(* PLC project Unnamed, Unknown Unnamed 1 *)
(* stored: creationDateTime 2026-07-02T15:04:41, modificationDateTime 2026-07-02T15:04:41 *)

FUNCTION DIV : ANY_NUM
  VAR_INPUT
    IN1 : ANY_NUM;
    IN2 : ANY_NUM;
  END_VAR

END_FUNCTION

FUNCTION MOVE : ANY
  VAR_INPUT
    IN : ANY;
  END_VAR

END_FUNCTION

PROGRAM main
  VAR_INPUT
    S1_LiDAR_Posisi : BOOL;  (* TRUE jika LiDAR mendeteksi posisi truk sudah pas/pas di tengah. *)
    S2_LoadCell_Stable : BOOL;  (* TRUE jika pembacaan berat dari load cell sudah stabil (tidak fluktuatif). *)
    Reset_Button : BOOL;  (* Tombol untuk meriset sistem setelah truk selesai ditimbang dan keluar. *)
    LiDAR_Volume_Raw : INT;  (* Data raw volume dari LiDAR. *)
    LoadCell_Weight_Raw : INT;  (* Data raw berat dari Load Cell. *)
  END_VAR
  VAR_OUTPUT
    Sistem_Ready : BOOL;  (* Lampu indikator jembatan timbang siap menerima truk. *)
    Alarm_Posisi : BOOL;  (* Lampu/sirine jika truk berhenti di posisi yang salah. *)
    Density_Result : REAL;  (* Hasil akhir perhitungan massa jenis (p). *)
  END_VAR
  VAR
    Lock_Data : BOOL;  (* Relay internal untuk mengunci proses kalkulasi. *)
    Volume_Locked : REAL;  (* Memori untuk menyimpan data volume yang sudah dikunci. *)
    Weight_Locked : REAL;  (* Memori untuk menyimpan data berat yang sudah dikunci. *)
  END_VAR
  VAR  (* added by the conversion: wires and edge detectors of the diagram *)
    R_TRIG1 : R_TRIG;
    R_TRIG2 : R_TRIG;
  END_VAR

(* LD diagram, written out as Structured Text *)
Sistem_Ready := NOT Lock_Data;
Alarm_Posisi := NOT S1_LiDAR_Posisi;
Lock_Data := (Lock_Data OR S1_LiDAR_Posisi AND S2_LoadCell_Stable) AND NOT Reset_Button;
R_TRIG1(CLK := Lock_Data);
IF R_TRIG1.Q THEN Volume_Locked := LiDAR_Volume_Raw; END_IF;
R_TRIG2(CLK := Lock_Data);
IF R_TRIG2.Q THEN Weight_Locked := LoadCell_Weight_Raw; END_IF;
IF Lock_Data THEN Density_Result := Weight_Locked / Volume_Locked; END_IF;
END_PROGRAM

CONFIGURATION Config0
  RESOURCE Res0 ON PLC
    TASK task0(INTERVAL := T#20ms, PRIORITY := 1);
    PROGRAM instance0 WITH task0 : main;
  END_RESOURCE
END_CONFIGURATION
